FUNCTION_BLOCK FB_OnOffTimer
VAR_INPUT
	tTimeOff	: TIME;
	tTimeOn		: TIME;
	nSpeedOn	: WORD;
	nSpeedOff	: WORD;
END_VAR
VAR_OUTPUT
	nSpeedOut	: WORD;
END_VAR
VAR
	TimerOff: TON;
	TimerOn: TOF;
END_VAR

TimerOff(IN:= NOT(TimerOn.Q), PT:= tTimeOff, Q=> TimerOn.IN, ET=> );
TimerOn(IN:= , PT:= tTimeOn, Q=> , ET=> );
IF TimerOn.Q THEN
	nSpeedOut := nSpeedOn;
	ELSE nSpeedOut := nSpeedOff;
END_IF

END_FUNCTION_BLOCK

(* stored: Version 1.1.0.1, ProductVersion 3.1.4022.18
   POU FB_OnOffTimer: Id {a7c94907-8f78-434d-b77b-1923a95ec5ca}, SpecialFunc None *)
